FUNCTION_BLOCK Test_AssertEquals_LREAL EXTENDS TUnitTestBase
VAR
    AssertionUnderTest : TAssertion(AssertionListenerMock);
    AssertionListenerMock : TAssertionListenerMock;
    LREAL_Variable : LREAL := 1.111;
END_VAR

// Initialise the classes under test (may be repaeting the tests)...
AssertionListenerMock.fb_Init(
    bInitRetains      := FALSE,
	bInCopyCode       := FALSE);
AssertionUnderTest.fb_Init(
    bInitRetains      := FALSE,
	bInCopyCode       := FALSE,
    AssertionListener := AssertionListenerMock);

// Test the assertion...
AssertionUnderTest.AssertEquals_LREAL(
    Expected := 2.222,
    Actual   := LREAL_Variable,
    Delta    := 0.001,
    VariableName := 'LREAL_Variable');
   
// Check the assertion worked...    
Assertion.AssertEquals_BOOL(
    Expected := TRUE,
    Actual   := AssertionListenerMock.AssertionFailed,
    VariableName := 'AssertionListenerMock.AssertionFailed');

// Check the assertion messages...    
Assertion.AssertEquals_STRING(
    Expected := 'AssertEquals_LREAL failed in AssertionListenerMock: Value "LREAL_Variable"',
    Actual   := AssertionListenerMock.AssertionMessage,
    VariableName := 'AssertionListenerMock.AssertionMessage');

Assertion.AssertEquals_STRING(
    Expected := '  Expected = 2.222000',
    Actual   := AssertionListenerMock.ExpectedAsString,
    VariableName := 'AssertionListenerMock.ExpectedAsString');

Assertion.AssertEquals_STRING(
    Expected := '  Actual   = 1.111000',
    Actual   := AssertionListenerMock.ActualAsString,
    VariableName := 'AssertionListenerMock.ActualAsString');

TestFinished();

END_FUNCTION_BLOCK

(* stored: Version 1.1.0.1, ProductVersion 3.1.4024.4
   POU Test_AssertEquals_LREAL: Id {b4c43a61-08cd-4fe8-b503-1f64bf7cdb15}, SpecialFunc None *)
